// TIA Portal V19 export
DATA_BLOCK "Module Diagnostic Result"   // DB59
{ S7_Optimized_Access := 'TRUE' }
// stored: AutoNumber false, MemoryReserve 0
   VAR RETAIN
      "2_AL1103" : Struct
         ErrorValue : Int;   // Error text/value
         ErrorCount : Int;   // How many times errors have occurred
         ErrorTime : DInt;   // Time since last error change
      END_STRUCT;
      "3_AL1307" : Struct
         ErrorValue : Int;   // Error text/value
         ErrorCount : Int;   // How many times errors have occurred
         ErrorTime : DInt;   // Time since last error change
      END_STRUCT;
      "4_AL1307" : Struct
         ErrorValue : Int;   // Error text/value
         ErrorCount : Int;   // How many times errors have occurred
         ErrorTime : DInt;   // Time since last error change
      END_STRUCT;
      "5_AL1307" : Struct
         ErrorValue : Int;   // Error text/value
         ErrorCount : Int;   // How many times errors have occurred
         ErrorTime : DInt;   // Time since last error change
      END_STRUCT;
      "6_AL1307" : Struct
         ErrorValue : Int;   // Error text/value
         ErrorCount : Int;   // How many times errors have occurred
         ErrorTime : DInt;   // Time since last error change
      END_STRUCT;
      "7_AL1307" : Struct
         ErrorValue : Int;   // Error text/value
         ErrorCount : Int;   // How many times errors have occurred
         ErrorTime : DInt;   // Time since last error change
      END_STRUCT;
      "8_Promag300" : Struct
         ErrorValue : Int;   // Error text/value
         ErrorCount : Int;   // How many times errors have occurred
         ErrorTime : DInt;   // Time since last error change
      END_STRUCT;
      "9_SinaG120" : Struct
         ErrorValue : Int;   // Error text/value
         ErrorCount : Int;   // How many times errors have occurred
         ErrorTime : DInt;   // Time since last error change
      END_STRUCT;
      "10_AL1307" : Struct
         ErrorValue : Int;   // Error text/value
         ErrorCount : Int;   // How many times errors have occurred
         ErrorTime : DInt;   // Time since last error change
      END_STRUCT;
      "11_PNCoup" : Struct
         ErrorValue : Int;   // Error text/value
         ErrorCount : Int;   // How many times errors have occurred
         ErrorTime : DInt;   // Time since last error change
      END_STRUCT;
      "12_AL1307" : Struct
         ErrorValue : Int;   // Error text/value
         ErrorCount : Int;   // How many times errors have occurred
         ErrorTime : DInt;   // Time since last error change
      END_STRUCT;
   END_VAR
BEGIN
END_DATA_BLOCK
